// TIA Portal V15.1 export
// export: Created 2024-05-17T05:38:29.667084Z, ExportSetting WithDefaults, DisplayName Totally Integrated Automation Portal, DisplayVersion V15.1 Update 5, DisplayName TIA Portal Openness, DisplayVersion V15.1 Update 5, DisplayName SINAMICS Startdrive Advanced, DisplayVersion V15.1, DisplayName G130, G150, S120, S150, SINAMICS MV, S210, DisplayVersion V15.1, DisplayName G110M, G120, G120C, G120D, G120P, DisplayVersion V15.1, DisplayName STEP 7 Professional, DisplayVersion V15.1 Update 5, DisplayName STEP 7 Safety, DisplayVersion V15.1, DisplayName WinCC Professional, DisplayVersion V15.1 Update 5, DisplayName SIMATIC Visualization Architect, DisplayVersion V15.1
FUNCTION_BLOCK "LPNIODiagMACS7-1500"   // FB2212, SCL
{ S7_Optimized_Access := 'TRUE' }
VERSION : 0.1
// stored: AutoNumber false, IsIECCheckEnabled false, IsRetainMemResEnabled false, MemoryReserve 100, SetENOAutomatically False, UDAEnableTagReadback false
   VAR_INPUT
      I_StartFillList { ExternalAccessible := 'False'; ExternalVisible := 'False'; ExternalWritable := 'False'} : Bool;
      I_LastDeviceNumber { ExternalAccessible := 'False'; ExternalVisible := 'False'; ExternalWritable := 'False'} : Int;   // Last Device of ProfiNet System
   END_VAR
   VAR_OUTPUT
      O_Done { ExternalAccessible := 'False'; ExternalVisible := 'False'; ExternalWritable := 'False'} : Bool;
      O_MACAddress { ExternalAccessible := 'False'; ExternalVisible := 'False'; ExternalWritable := 'False'} : Array[0..255] of String[18];
   END_VAR
   VAR_IN_OUT
      IO_DeviceExist : Array[0..255] of Bool;   // IO devices exist
      IO_HWIdentifier : Array[0..255] of UInt;   // HW Device
      IO_GetStationMAC : Array[0..255] of IF_CONF_MAC;   // Read out Station Information
   END_VAR
   VAR
      Index { ExternalAccessible := 'False'; ExternalVisible := 'False'; ExternalWritable := 'False'} : Int;
      LastDeviceNumber { ExternalAccessible := 'False'; ExternalVisible := 'False'; ExternalWritable := 'False'} : Int;   // Last Device of ProfiNet System
      Done { ExternalAccessible := 'False'; ExternalVisible := 'False'; ExternalWritable := 'False'} : Bool;
      DoneDelay { ExternalAccessible := 'False'; ExternalVisible := 'False'; ExternalWritable := 'False'} : Bool;
      ReturnGetStationInfoBusy_MAC { ExternalAccessible := 'False'; ExternalVisible := 'False'; ExternalWritable := 'False'} : Bool;   // Temp
      ReturnGetStationInfoDone_MAC { ExternalAccessible := 'False'; ExternalVisible := 'False'; ExternalWritable := 'False'} : Bool;   // Temp
      ReturnGetStationInfoError_MAC { ExternalAccessible := 'False'; ExternalVisible := 'False'; ExternalWritable := 'False'} : Bool;   // Temp
      ReturnGetStationInfoStatus_MAC { ExternalAccessible := 'False'; ExternalVisible := 'False'; ExternalWritable := 'False'} : Word;   // Temp
      MACAddress_ADDR1 { ExternalAccessible := 'False'; ExternalVisible := 'False'; ExternalWritable := 'False'} : String[2];
      MACAddress_ADDR2 { ExternalAccessible := 'False'; ExternalVisible := 'False'; ExternalWritable := 'False'} : String[2];
      MACAddress_ADDR3 { ExternalAccessible := 'False'; ExternalVisible := 'False'; ExternalWritable := 'False'} : String[2];
      MACAddress_ADDR4 { ExternalAccessible := 'False'; ExternalVisible := 'False'; ExternalWritable := 'False'} : String[2];
      MACAddress_ADDR5 { ExternalAccessible := 'False'; ExternalVisible := 'False'; ExternalWritable := 'False'} : String[2];
      MACAddress_ADDR6 { ExternalAccessible := 'False'; ExternalVisible := 'False'; ExternalWritable := 'False'} : String[2];
      MACAddress { ExternalAccessible := 'False'; ExternalVisible := 'False'; ExternalWritable := 'False'} : String[18];
      RetVal { ExternalAccessible := 'False'; ExternalVisible := 'False'; ExternalWritable := 'False'} : Word;
      GetStationInfo_MAC { ExternalAccessible := 'False'; ExternalVisible := 'False'; ExternalWritable := 'False'; S7_SetPoint := 'True'} : GetStationInfo;
      TimerDone { ExternalAccessible := 'False'; ExternalVisible := 'False'; ExternalWritable := 'False'; S7_SetPoint := 'True'} : TON_TIME;
      EdgeStartFillList { ExternalAccessible := 'False'; ExternalVisible := 'False'; ExternalWritable := 'False'; S7_SetPoint := 'True'} : R_TRIG;
   END_VAR
BEGIN
   #EdgeStartFillList(CLK := #I_StartFillList);

   IF #EdgeStartFillList.Q THEN
       #Done := False;
       #Index := 0;
   END_IF;

   #LastDeviceNumber := #I_LastDeviceNumber;
   IF #I_LastDeviceNumber < 1 THEN
       #LastDeviceNumber := 1;
   END_IF;
   IF #I_LastDeviceNumber > 254 THEN
       #LastDeviceNumber := 254;
   END_IF;

   #TimerDone(IN := #Done,
              PT := T#500ms,
              Q => #DoneDelay);

   IF (#I_StartFillList & NOT #Done) THEN
       #Index := #Index + 1;
       WHILE (#IO_DeviceExist[#Index] & NOT #ReturnGetStationInfoDone_MAC) DO
           #GetStationInfo_MAC(REQ := #IO_DeviceExist[#Index] & NOT #ReturnGetStationInfoBusy_MAC,
               LADDR := #IO_HWIdentifier[#Index],
               MODE := 2,
               DONE => #ReturnGetStationInfoDone_MAC,
               BUSY => #ReturnGetStationInfoBusy_MAC,
               ERROR => #ReturnGetStationInfoError_MAC,
               STATUS => #ReturnGetStationInfoStatus_MAC,
               DATA := #IO_GetStationMAC[#Index]);
       END_WHILE;
       #ReturnGetStationInfoDone_MAC := False;

       #RetVal := HTA(IN := #IO_GetStationMAC[#Index].Mac[1], N := 2, OUT => #MACAddress_ADDR1);
       #RetVal := HTA(IN := #IO_GetStationMAC[#Index].Mac[2], N := 2, OUT => #MACAddress_ADDR2);
       #RetVal := HTA(IN := #IO_GetStationMAC[#Index].Mac[3], N := 2, OUT => #MACAddress_ADDR3);
       #RetVal := HTA(IN := #IO_GetStationMAC[#Index].Mac[4], N := 2, OUT => #MACAddress_ADDR4);
       #RetVal := HTA(IN := #IO_GetStationMAC[#Index].Mac[5], N := 2, OUT => #MACAddress_ADDR5);
       #RetVal := HTA(IN := #IO_GetStationMAC[#Index].Mac[6], N := 2, OUT => #MACAddress_ADDR6);

       #MACAddress := CONCAT_STRING(IN1 := #MACAddress_ADDR1, IN2 := '.');
       #MACAddress := CONCAT_STRING(IN1 := #MACAddress, IN2 := #MACAddress_ADDR2);
       #MACAddress := CONCAT_STRING(IN1 := #MACAddress, IN2 := '.');
       #MACAddress := CONCAT_STRING(IN1 := #MACAddress, IN2 := #MACAddress_ADDR3);
       #MACAddress := CONCAT_STRING(IN1 := #MACAddress, IN2 := '.');
       #MACAddress := CONCAT_STRING(IN1 := #MACAddress, IN2 := #MACAddress_ADDR4);
       #MACAddress := CONCAT_STRING(IN1 := #MACAddress, IN2 := '.');
       #MACAddress := CONCAT_STRING(IN1 := #MACAddress, IN2 := #MACAddress_ADDR5);
       #MACAddress := CONCAT_STRING(IN1 := #MACAddress, IN2 := '.');
       #MACAddress := CONCAT_STRING(IN1 := #MACAddress, IN2 := #MACAddress_ADDR6);
       #O_MACAddress[#Index] := #MACAddress;
       IF #Index = #LastDeviceNumber THEN
           #Done := True;
       END_IF;
   END_IF;

   #O_Done := #DoneDelay;
END_FUNCTION_BLOCK
